{region '#Template'}
	{attribute 'Version' := '1.2.1.0'}
	{attribute 'Tags' := '"LCID": "1031", "Text": "Universal, Analog, Aggregate"'}
	{attribute 'Tags' := '"LCID": "1033", "Text": "Universal, Analog, Aggregate"'}
	{attribute 'Using' := '"Type": "Template", "URI": "EC_AMEV"'}
	{attribute 'Using' := '"Type": "Template", "URI": "BA2_Param"'}
	{attribute 'Description' := '"LCID": "1031", "Text": "Aktor binär"'}
	{attribute 'Description' := '"LCID": "1033", "Text": "Actuator binary"'}
{endregion}
FUNCTION_BLOCK FB_BA_ActuatorCmd EXTENDS FB_BA_AggregateB
VAR_OUTPUT
	bCmd							: BOOL;
END_VAR
VAR_INPUT CONSTANT
	Cmd						: FB_BA_BO_IO;			
END_VAR

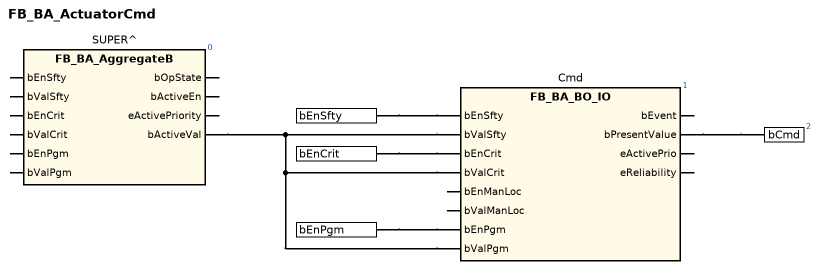
SUPER^(); // FB_BA_AggregateB
Cmd(
    bEnSfty := bEnSfty,
    bValSfty := SUPER^.bActiveVal,
    bEnCrit := bEnCrit,
    bValCrit := SUPER^.bActiveVal,
    bEnPgm := bEnPgm,
    bValPgm := SUPER^.bActiveVal); // FB_BA_BO_IO
bCmd := Cmd.bPresentValue;

METHOD FB_init : BOOL
VAR_INPUT
	bInitRetains : BOOL; // if TRUE, the retain variables are initialized (warm start / cold start)
	bInCopyCode : BOOL;  // if TRUE, the instance afterwards gets moved into the copy code (online change)
END_VAR
Cmd.iParent							:= THIS^;
Cmd.iLabel							:= LblUniFieldDevice.Aggregat_Cmd;			
Cmd.sObjectName						:= '{Idx=01}';	
Cmd.sDeviceType						:= '';
Cmd.bEnOutOfService					:= FALSE;
Cmd.ePolarity						:= E_BA_Polarity.eNormal;
Cmd.eFeedbackPolarity				:= E_BA_Polarity.eNormal;
Cmd.eOverriddenPolarity				:= E_BA_Polarity.eReverse;
Cmd.sActiveText 					:= txtEvent_On;
Cmd.sInactiveText 					:= txtEvent_Off;
Cmd.nStateChangeCount				:= 0;
Cmd.nActiveTimeElapsed				:= 0;
Cmd.nMinimumOnTime					:= 0;
Cmd.nMinimumOffTime					:= 0;
Cmd.bEnManualRm						:= FALSE;	//	Priority  8	
Cmd.bValManualRm					:= FALSE;	//	Priority  8
Cmd.bDefaultValue					:= FALSE;
Cmd.nEventClassID					:= EC_ID.NC40;
Cmd.stTimeDelay.nToNormal			:= BA2_Param.nDefTimeDelay_ToNormal;
Cmd.stTimeDelay.nToAbnormal			:= BA2_Param.nDefTimeDelay_ToAbnormal;
Cmd.bAcknowledgeRm					:= FALSE;		
Cmd.aEventTransitionText[1]			:= txtEvent_Disturb;
Cmd.aEventTransitionText[2]			:= txtEvent_None;
Cmd.aEventTransitionText[3]			:= txtEvent_Normal;
Cmd.bEventDetectionEnable			:= FALSE;
Cmd.aEventEnable[1]					:= TRUE;			//	to_offnormal
Cmd.aEventEnable[2]					:= TRUE;			//	to_fault
Cmd.aEventEnable[3]					:= TRUE;			//	to_normal
Cmd.eEnPlantLock					:= E_BA_LockPriority.eNoLock;
END_METHOD

END_FUNCTION_BLOCK

(* stored: Version 1.1.0.1, ProductVersion 3.1.4024.9
   POU FB_BA_ActuatorCmd: Id {1c219490-3f24-42eb-b20a-f4bdb1f26090}, SpecialFunc None
   Method FB_init: Id {ec100382-c238-4fed-a08f-633c3f6ce638} *)
